PROGRAM MAIN
VAR

END_VAR


	P_SortingConveyor_proceduralApproach();

END_PROGRAM

(* stored: Version 1.1.0.1, ProductVersion 3.1.4024.12
   POU MAIN: Id {d83b5889-783a-434a-87bd-f33de96679bb}, SpecialFunc None *)
